TYPE DUT_SERVER_SKILL_INPUT :
STRUCT
	///Range of parameters
	ParameterInput: DUT_SERVER_PARAMETERINPUTARRAY;
	///Start process
	Execute: BOOL;
END_STRUCT
END_TYPE

(* stored: Version 1.1.0.1, ProductVersion 3.1.0.25
   DUT DUT_SERVER_SKILL_INPUT: Id {db92dc5d-1623-456f-852c-06ab20b7eb28} *)
